TYPE ST_AdjustmentMotionConfig :
STRUCT
    stX : ST_VelocityConfig;
    stY : ST_VelocityConfig;
    stZ : ST_VelocityConfig;
    fPositionTolerance : LREAL;
    tMoveTimeout : TIME;
END_STRUCT
END_TYPE

(* stored: Version 1.1.0.1, ProductVersion 3.1.4026.20
   DUT ST_AdjustmentMotionConfig: Id {03da73f8-946f-42da-875f-e25aee363acc} *)
